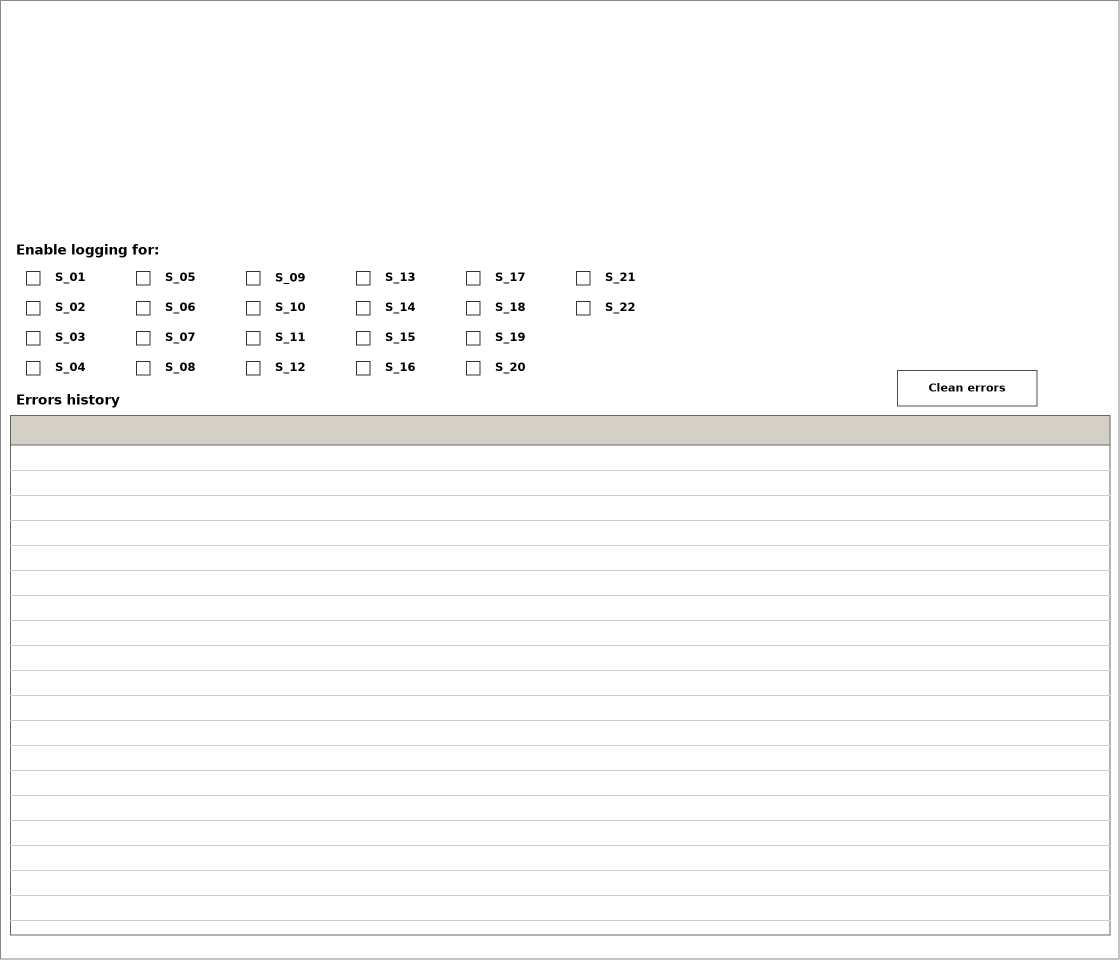
VISUALIZATION vErrorsData  // 1120x960
    Label (13,390 150x20), "Errors history"
    Rectangle (897,370 140x36), "Clean errors"
        OnMouseClick: execute { GVL.fbAlarmMasterTable.mReset(); }
    Checkbox (24,265 26x26), variable: GVL.abChoseStationsToLog[1]
    Label (52,265 49x24), "S_01"
    Label (13,240 214x20), "Enable logging for:"
    Checkbox (24,295 26x26), variable: GVL.abChoseStationsToLog[2]
    Label (52,295 49x24), "S_02"
    Checkbox (24,325 26x26), variable: GVL.abChoseStationsToLog[3]
    Label (52,325 49x24), "S_03"
    Checkbox (24,355 26x26), variable: GVL.abChoseStationsToLog[4]
    Label (52,355 49x24), "S_04"
    Checkbox (134,265 26x26), variable: GVL.abChoseStationsToLog[5]
    Label (162,265 49x24), "S_05"
    Label (162,295 49x24), "S_06"
    Checkbox (134,295 26x26), variable: GVL.abChoseStationsToLog[6]
    Label (162,325 49x24), "S_07"
    Checkbox (134,325 26x26), variable: GVL.abChoseStationsToLog[7]
    Label (162,355 49x24), "S_08"
    Checkbox (134,355 26x26), variable: GVL.abChoseStationsToLog[8]
    Checkbox (244,265 26x26), variable: GVL.abChoseStationsToLog[9]
    Label (272,266 49x23), "S_09"
    Checkbox (244,325 26x26), variable: GVL.abChoseStationsToLog[11]
    Label (272,325 49x24), "S_11"
    Checkbox (244,355 26x26), variable: GVL.abChoseStationsToLog[12]
    Label (272,355 49x24), "S_12"
    Checkbox (354,265 26x26), variable: GVL.abChoseStationsToLog[13]
    Label (382,265 49x24), "S_13"
    Checkbox (354,295 26x26), variable: GVL.abChoseStationsToLog[14]
    Label (382,295 49x24), "S_14"
    Label (382,325 49x24), "S_15"
    Checkbox (354,325 26x26), variable: GVL.abChoseStationsToLog[15]
    Label (382,355 49x24), "S_16"
    Checkbox (354,355 26x26), variable: GVL.abChoseStationsToLog[16]
    Label (492,265 49x24), "S_17"
    Checkbox (464,265 26x26), variable: GVL.abChoseStationsToLog[17]
    Checkbox (464,295 26x26), variable: GVL.abChoseStationsToLog[18]
    Label (492,295 49x24), "S_18"
    Checkbox (464,325 26x26), variable: GVL.abChoseStationsToLog[19]
    Label (492,325 49x24), "S_19"
    Checkbox (464,355 26x26), variable: GVL.abChoseStationsToLog[20]
    Label (492,355 49x24), "S_20"
    Checkbox (574,265 26x26), variable: GVL.abChoseStationsToLog[21]
    Label (602,265 49x24), "S_21"
    Checkbox (574,295 26x26), variable: GVL.abChoseStationsToLog[22]
    Label (602,295 49x24), "S_22"
    Checkbox (244,295 26x26), variable: GVL.abChoseStationsToLog[10]
    Label (272,295 49x24), "S_10"
    Table (10,415 1100x520), data array: GVL.fbAlarmMasterTable.astErrTable
        p1128707560: GVL.fbAlarmMasterTable.uiRowNumber
        p3854506369: GVL.fbAlarmMasterTable.astErrTable[INDEX].dtEventTime
        p1892666644: GVL.fbAlarmMasterTable.astErrTable[INDEX].sMachineId
        p338671338: GVL.fbAlarmMasterTable.astErrTable[INDEX].sEventDescription
        p2170511999: GVL.fbAlarmMasterTable.astErrTable[INDEX].dwErrorCode
        p3723444502: GVL.fbAlarmMasterTable.astErrTable[INDEX].uiRepeatQty
        p1218418051: GVL.fbAlarmMasterTable.astErrTable[INDEX].nAlarmClass
        p2232123230: Event time
        p511219082: Machine ID
        p1755163831: Event description
        p4092479075: Error Code
        p2237128397: Repeat Qty
END_VISUALIZATION

(* stored: Version 1.1.0.1, ProductVersion 3.1.4024.12
   Visu vErrorsData: Id {71071bd0-cfd0-4512-9805-315244616f96} *)
